{attribute 'qualified_only'}
{attribute 'strict'}
{attribute 'to_string'}
TYPE E_MoveState :
(
    IDLING:=0,
    INIT_MOVE:=10,
    START_MOVE:=20,
    MOVE_IN_PROGRESS :=30,
    TARGET_REACHED:=40,
    MOVE_INTERRUPTED:=50,
    MOVE_ABORTED:=60,
    MOVE_DONE:=70,
    MOVE_ERROR:=-99
);
END_TYPE

(* stored: Version 1.1.0.1
   DUT E_MoveState: Id {933b85d6-53dd-4c3d-b3b1-3a89b00aa8fa} *)
